// SIMATIC S7-200 project (STEP 7-Micro/WIN), CPU 224 REL 02.01

SYMBOL_TABLE USER1
went             VW140
ogrz             VW130
tz               VW120
h                VW110
ta               VW100
T                AIW8
Spoczynek        Q0.1
Ogrzewanie       Q0.2
Wentylacja       Q0.0
TZwiecej         I0.1
TZmniej          I0.2
TZreset          I0.3
hwiecej          I0.4
hmniej           I0.5
hreset           I0.6
END_SYMBOL_TABLE

ORGANIZATION_BLOCK MAIN:OB1
TITLE=
BEGIN
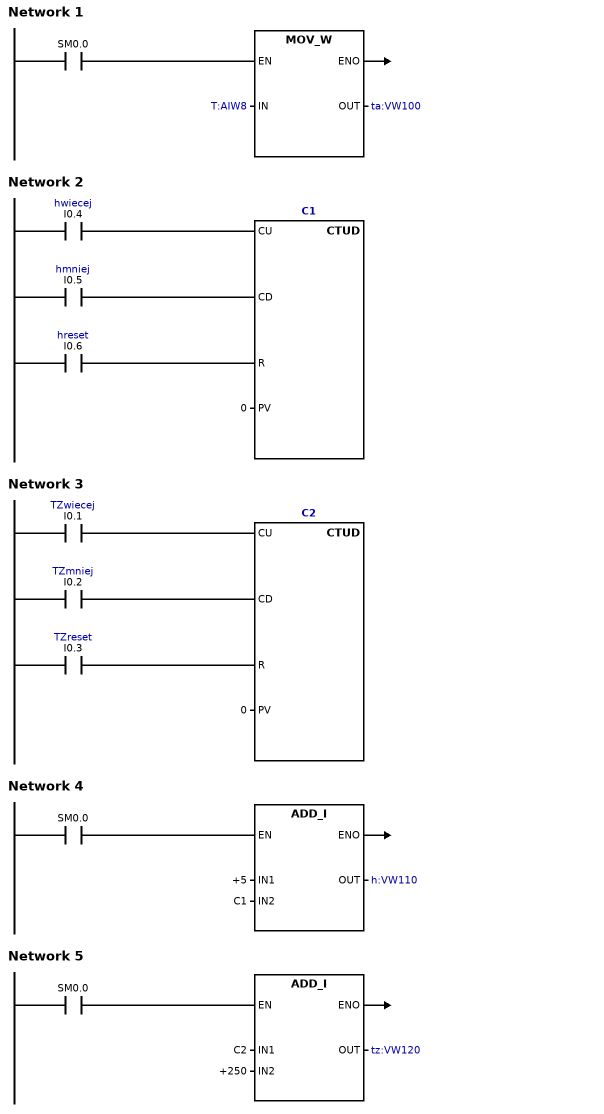
Network 1
LD     SM0.0
MOVW   T:AIW8, ta:VW100
Network 2
LD     hwiecej:I0.4
LD     hmniej:I0.5
LD     hreset:I0.6
CTUD   C1, 0
Network 3
LD     TZwiecej:I0.1
LD     TZmniej:I0.2
LD     TZreset:I0.3
CTUD   C2, 0
Network 4
LD     SM0.0
MOVW   +5, h:VW110
+I     C1, h:VW110
Network 5
LD     SM0.0
MOVW   C2, tz:VW120
+I     +250, tz:VW120
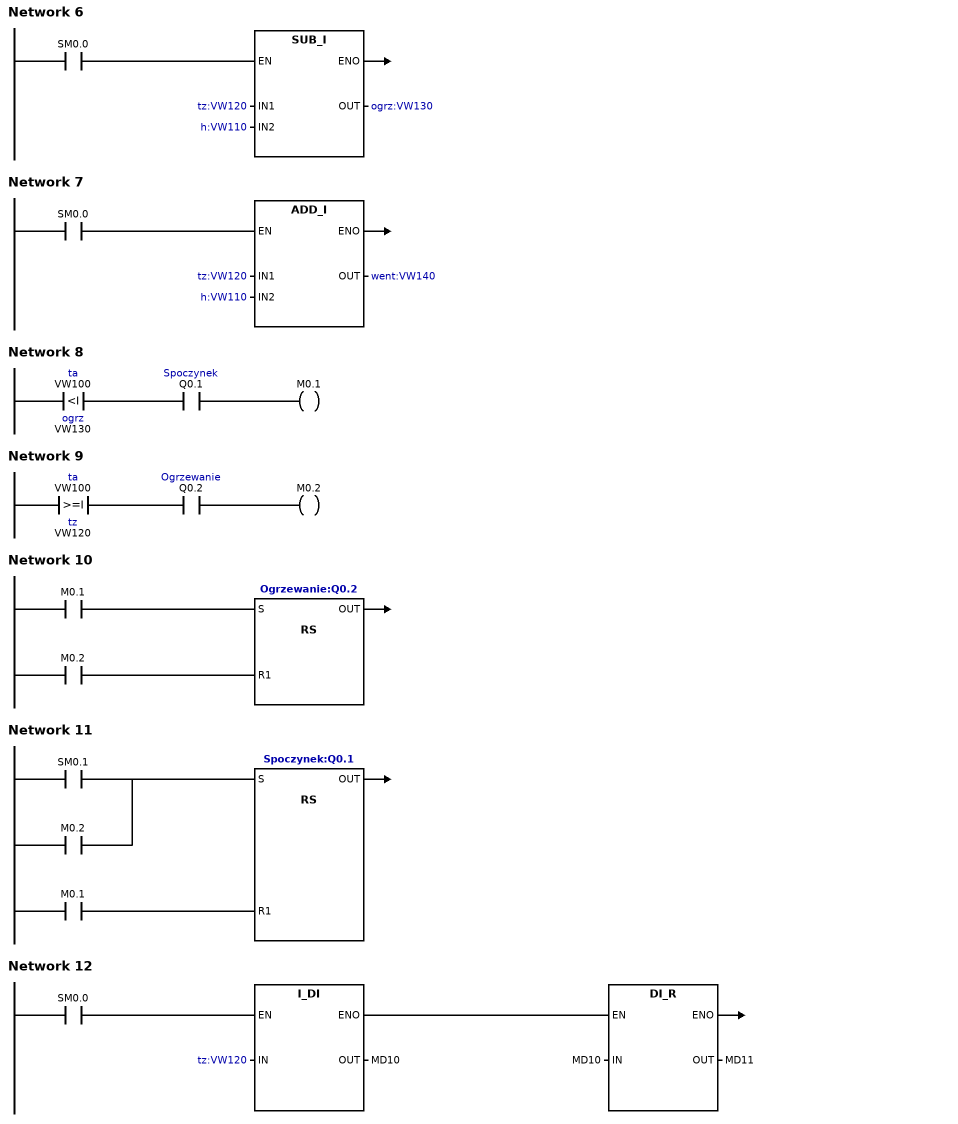
Network 6
LD     SM0.0
MOVW   tz:VW120, ogrz:VW130
-I     h:VW110, ogrz:VW130
Network 7
LD     SM0.0
MOVW   tz:VW120, went:VW140
+I     h:VW110, went:VW140
Network 8
LDW<   ta:VW100, ogrz:VW130
A      Spoczynek:Q0.1
=      M0.1
Network 9
LDW>=  ta:VW100, tz:VW120
A      Ogrzewanie:Q0.2
=      M0.2
Network 10
LD     M0.1
LD     M0.2
NOT
LPS
A      Ogrzewanie:Q0.2
=      Ogrzewanie:Q0.2
LPP
ALD
O      Ogrzewanie:Q0.2
=      Ogrzewanie:Q0.2
Network 11
LD     SM0.1
O      M0.2
LD     M0.1
NOT
LPS
A      Spoczynek:Q0.1
=      Spoczynek:Q0.1
LPP
ALD
O      Spoczynek:Q0.1
=      Spoczynek:Q0.1
Network 12
// (network saved uncompiled; LAD cells follow)
// row 0: c0 -| |- SM0.0  c1 --  c2 [I_DI EN:=power@row0, IN:=tz:VW120, ENO=>power, OUT=>MD10]  c3 --  c4 --  c5 [DI_R EN:=power@row0, IN:=MD10, ENO=>power, OUT=>MD11]  c6 ->
// row 1: c2 [box]  c5 [box]
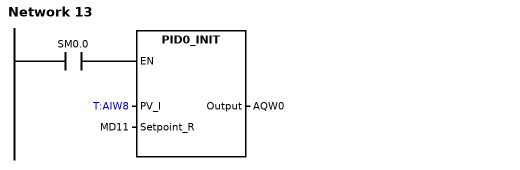
Network 13
// (network saved uncompiled; LAD cells follow)
// row 0: c0 -| |- SM0.0  c1 [PID0_INIT EN:=power@row0, PV_I:=T:AIW8, Setpoint_R:=MD11, Output=>AQW0]
// row 1: c1 [box]
END_ORGANIZATION_BLOCK

// SBR1: protected block, not included

// INT1: protected block, not included

// (further data pages could not be read)
